FUNCTION_BLOCK PERCENT_AJUST (* Sets a percentual value from a given input *)
  (* Standard: 61499-2 *)
  (* Version 1.0, 09-01-12, Guilherme Jarentchuk, Universidade do Estado de Santa Catarina *)
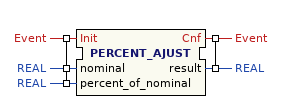
  EVENT_INPUT
    Init WITH nominal, percent_of_nominal; (* Initialize execution *)
  END_EVENT
  EVENT_OUTPUT
    Cnf WITH result; (* Confirm execution *)
  END_EVENT
  VAR_INPUT
    nominal : REAL;
    percent_of_nominal : REAL := 100;
  END_VAR
  VAR_OUTPUT
    result : REAL;
  END_VAR
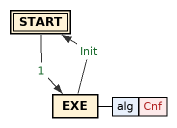
  EC_STATES
    START;
    EXE : alg -> Cnf;
  END_STATES
  EC_TRANSITIONS
    START TO EXE := 1;
    EXE TO START := Init;
  END_TRANSITIONS
  ALGORITHM alg IN Lua:
result = nominal*(percent_of_nominal/100)
  END_ALGORITHM
END_FUNCTION_BLOCK
